% RSLogix 500 project Temperature Control and Alarm System.RSS, saved by version 8.30.00.16 %
PROJECT "UNTITLED"    % processor: Bul.1763 MicroLogix 1100 Series B %

PROGRAM FILES
  LAD 2 "MAIN"  9 rungs
  LAD 3 "DIGITAL IO"  10 rungs
  LAD 4 "ANALOG IO"  4 rungs
  LAD 5 "MANUAL"  10 rungs
  LAD 6 "AUTOMATIC"  3 rungs
  LAD 7 "ALARMS"  13 rungs
  LAD 8 "TEMP PID"  10 rungs
  LAD 9 "PROCESS"  9 rungs
  LAD 10 "TIMERS"  7 rungs

DATA FILES
  O0 OUTPUT  4 elements
  I1 INPUT  6 elements
  S2 STATUS  66 elements
  B3 BINARY  3 elements
  T4 TIMER  6 elements
  C5 COUNTER  1 elements
  R6 CONTROL  1 elements
  N7 INTEGER  5 elements
  F8 FLOAT  6 elements

LADDER 2 "MAIN"
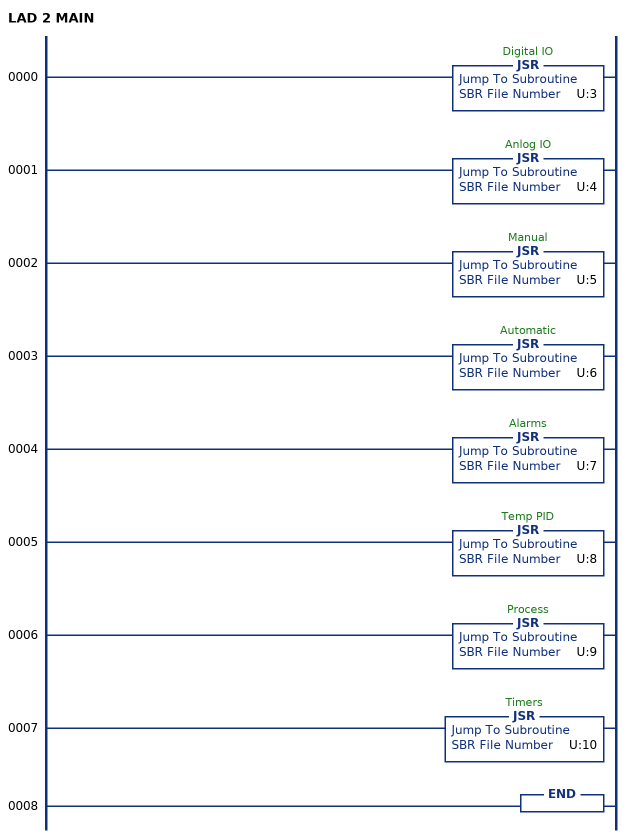
% Rung: 0 %
SOR JSR U:3 EOR
%   U:3  "Digital IO" %
% Rung: 1 %
SOR JSR U:4 EOR
%   U:4  "Anlog IO" %
% Rung: 2 %
SOR JSR U:5 EOR
%   U:5  "Manual" %
% Rung: 3 %
SOR JSR U:6 EOR
%   U:6  "Automatic" %
% Rung: 4 %
SOR JSR U:7 EOR
%   U:7  "Alarms" %
% Rung: 5 %
SOR JSR U:8 EOR
%   U:8  "Temp PID" %
% Rung: 6 %
SOR JSR U:9 EOR
%   U:9  "Process" %
% Rung: 7 %
SOR JSR U:10 EOR
%   U:10  "Timers" %
% Rung: 8 %
SOR END EOR

LADDER 3 "DIGITAL IO"
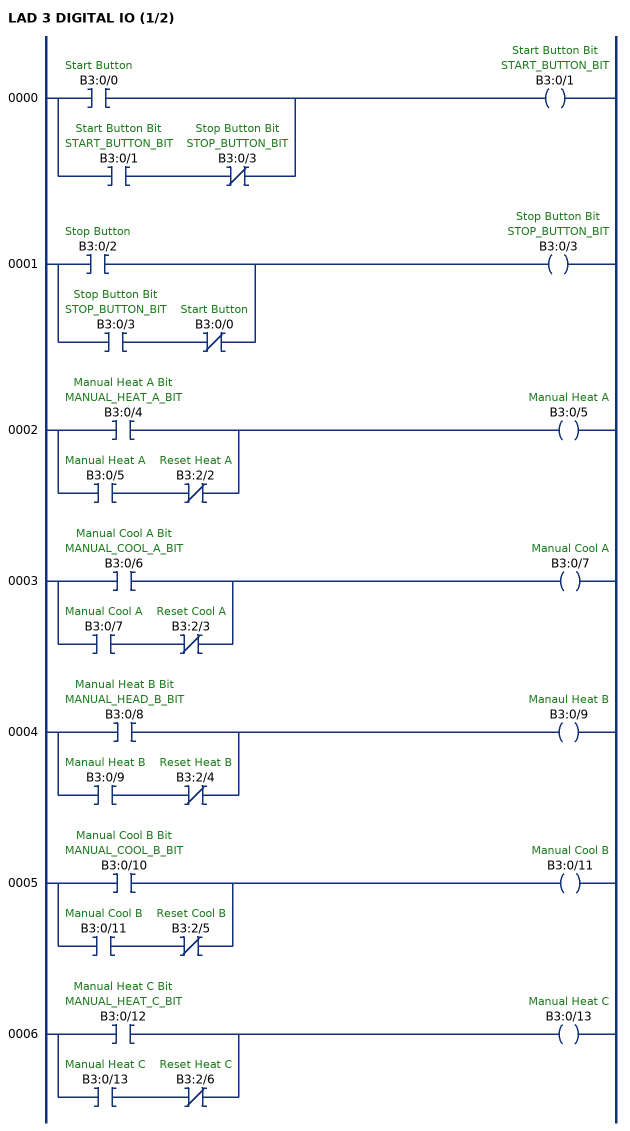
% Rung: 0 %
SOR BST XIC B3:0/0 NXB XIC B3:0/1 XIO B3:0/3 BND OTE B3:0/1 EOR
%   B3:0/0  "Start Button" %
%   B3:0/1  START_BUTTON_BIT  "Start Button Bit" %
%   B3:0/3  STOP_BUTTON_BIT  "Stop Button Bit" %
% Rung: 1 %
SOR BST XIC B3:0/2 NXB XIC B3:0/3 XIO B3:0/0 BND OTE B3:0/3 EOR
%   B3:0/2  "Stop Button" %
%   B3:0/3  STOP_BUTTON_BIT  "Stop Button Bit" %
%   B3:0/0  "Start Button" %
% Rung: 2 %
SOR BST XIC B3:0/4 NXB XIC B3:0/5 XIO B3:2/2 BND OTE B3:0/5 EOR
%   B3:0/4  MANUAL_HEAT_A_BIT  "Manual Heat A Bit" %
%   B3:0/5  "Manual Heat A" %
%   B3:2/2  "Reset Heat A" %
% Rung: 3 %
SOR BST XIC B3:0/6 NXB XIC B3:0/7 XIO B3:2/3 BND OTE B3:0/7 EOR
%   B3:0/6  MANUAL_COOL_A_BIT  "Manual Cool A Bit" %
%   B3:0/7  "Manual Cool A" %
%   B3:2/3  "Reset Cool A" %
% Rung: 4 %
SOR BST XIC B3:0/8 NXB XIC B3:0/9 XIO B3:2/4 BND OTE B3:0/9 EOR
%   B3:0/8  MANUAL_HEAD_B_BIT  "Manual Heat B Bit" %
%   B3:0/9  "Manaul Heat B" %
%   B3:2/4  "Reset Heat B" %
% Rung: 5 %
SOR BST XIC B3:0/10 NXB XIC B3:0/11 XIO B3:2/5 BND OTE B3:0/11 EOR
%   B3:0/10  MANUAL_COOL_B_BIT  "Manual Cool B Bit" %
%   B3:0/11  "Manual Cool B" %
%   B3:2/5  "Reset Cool B" %
% Rung: 6 %
SOR BST XIC B3:0/12 NXB XIC B3:0/13 XIO B3:2/6 BND OTE B3:0/13 EOR
%   B3:0/12  MANUAL_HEAT_C_BIT  "Manual Heat C Bit" %
%   B3:0/13  "Manual Heat C" %
%   B3:2/6  "Reset Heat C" %

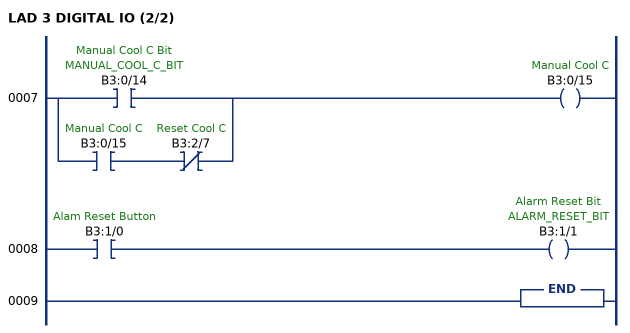
% Rung: 7 %
SOR BST XIC B3:0/14 NXB XIC B3:0/15 XIO B3:2/7 BND OTE B3:0/15 EOR
%   B3:0/14  MANUAL_COOL_C_BIT  "Manual Cool C Bit" %
%   B3:0/15  "Manual Cool C" %
%   B3:2/7  "Reset Cool C" %
% Rung: 8 %
SOR XIC B3:1/0 OTE B3:1/1 EOR
%   B3:1/0  "Alam Reset Button" %
%   B3:1/1  ALARM_RESET_BIT  "Alarm Reset Bit" %
% Rung: 9 %
SOR END EOR

LADDER 4 "ANALOG IO"
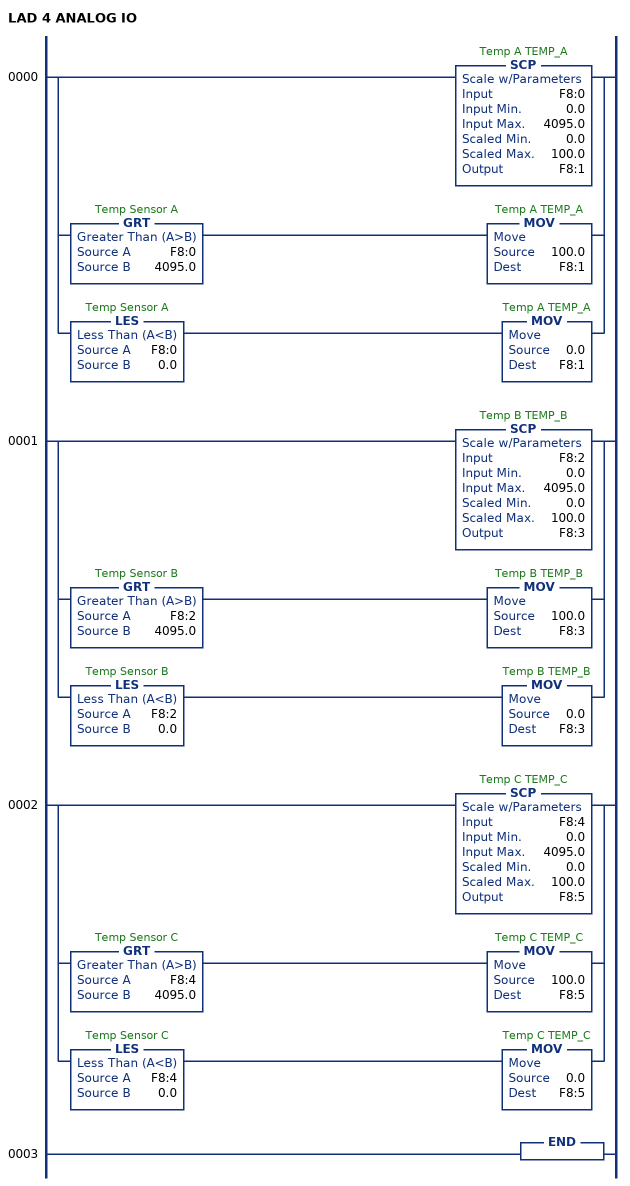
% Rung: 0 %
SOR BST BST SCP F8:0 0.0 4095.0 0.0 100.0 F8:1 NXB GRT F8:0 4095.0 MOV 100.0 F8:1 BND NXB LES F8:0 0.0 MOV 0.0 F8:1 BND EOR
%   F8:0  "Temp Sensor A" %
%   F8:1  TEMP_A  "Temp A" %
% Rung: 1 %
SOR BST BST SCP F8:2 0.0 4095.0 0.0 100.0 F8:3 NXB GRT F8:2 4095.0 MOV 100.0 F8:3 BND NXB LES F8:2 0.0 MOV 0.0 F8:3 BND EOR
%   F8:2  "Temp Sensor B" %
%   F8:3  TEMP_B  "Temp B" %
% Rung: 2 %
SOR BST BST SCP F8:4 0.0 4095.0 0.0 100.0 F8:5 NXB GRT F8:4 4095.0 MOV 100.0 F8:5 BND NXB LES F8:4 0.0 MOV 0.0 F8:5 BND EOR
%   F8:4  "Temp Sensor C" %
%   F8:5  TEMP_C  "Temp C" %
% Rung: 3 %
SOR END EOR

LADDER 5 "MANUAL"
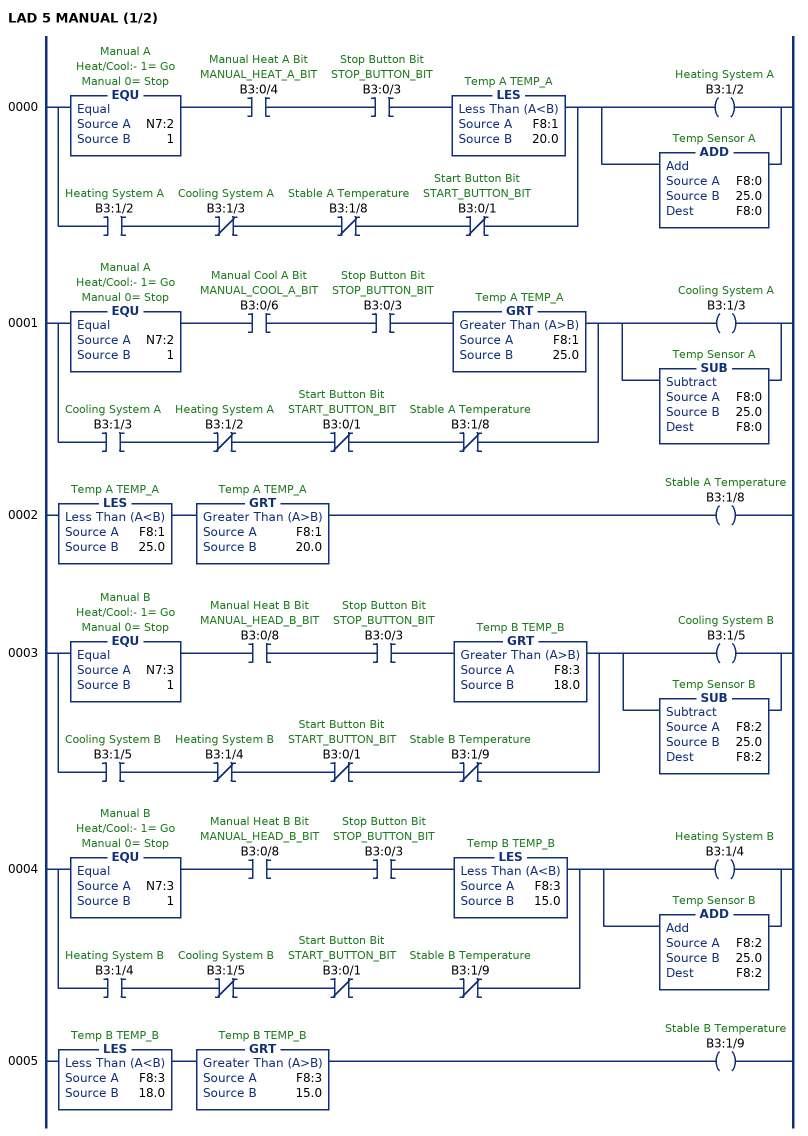
% Rung: 0 %
SOR BST EQU N7:2 1 XIC B3:0/4 XIC B3:0/3 LES F8:1 20.0 NXB XIC B3:1/2 XIO B3:1/3 XIO B3:1/8 XIO B3:0/1 BND BST OTE B3:1/2 NXB ADD F8:0 25.0 F8:0 BND EOR
%   N7:2  "Manual A Heat/Cool:- 1= Go Manual 0= Stop" %
%   B3:0/4  MANUAL_HEAT_A_BIT  "Manual Heat A Bit" %
%   B3:0/3  STOP_BUTTON_BIT  "Stop Button Bit" %
%   F8:1  TEMP_A  "Temp A" %
%   B3:1/2  "Heating System A" %
%   B3:1/3  "Cooling System A" %
%   B3:1/8  "Stable A Temperature" %
%   B3:0/1  START_BUTTON_BIT  "Start Button Bit" %
%   F8:0  "Temp Sensor A" %
% Rung: 1 %
SOR BST EQU N7:2 1 XIC B3:0/6 XIC B3:0/3 GRT F8:1 25.0 NXB XIC B3:1/3 XIO B3:1/2 XIO B3:0/1 XIO B3:1/8 BND BST OTE B3:1/3 NXB SUB F8:0 25.0 F8:0 BND EOR
%   N7:2  "Manual A Heat/Cool:- 1= Go Manual 0= Stop" %
%   B3:0/6  MANUAL_COOL_A_BIT  "Manual Cool A Bit" %
%   B3:0/3  STOP_BUTTON_BIT  "Stop Button Bit" %
%   F8:1  TEMP_A  "Temp A" %
%   B3:1/3  "Cooling System A" %
%   B3:1/2  "Heating System A" %
%   B3:0/1  START_BUTTON_BIT  "Start Button Bit" %
%   B3:1/8  "Stable A Temperature" %
%   F8:0  "Temp Sensor A" %
% Rung: 2 %
SOR LES F8:1 25.0 GRT F8:1 20.0 OTE B3:1/8 EOR
%   F8:1  TEMP_A  "Temp A" %
%   B3:1/8  "Stable A Temperature" %
% Rung: 3 %
SOR BST EQU N7:3 1 XIC B3:0/8 XIC B3:0/3 GRT F8:3 18.0 NXB XIC B3:1/5 XIO B3:1/4 XIO B3:0/1 XIO B3:1/9 BND BST OTE B3:1/5 NXB SUB F8:2 25.0 F8:2 BND EOR
%   N7:3  "Manual B Heat/Cool:- 1= Go Manual 0= Stop" %
%   B3:0/8  MANUAL_HEAD_B_BIT  "Manual Heat B Bit" %
%   B3:0/3  STOP_BUTTON_BIT  "Stop Button Bit" %
%   F8:3  TEMP_B  "Temp B" %
%   B3:1/5  "Cooling System B" %
%   B3:1/4  "Heating System B" %
%   B3:0/1  START_BUTTON_BIT  "Start Button Bit" %
%   B3:1/9  "Stable B Temperature" %
%   F8:2  "Temp Sensor B" %
% Rung: 4 %
SOR BST EQU N7:3 1 XIC B3:0/8 XIC B3:0/3 LES F8:3 15.0 NXB XIC B3:1/4 XIO B3:1/5 XIO B3:0/1 XIO B3:1/9 BND BST OTE B3:1/4 NXB ADD F8:2 25.0 F8:2 BND EOR
%   N7:3  "Manual B Heat/Cool:- 1= Go Manual 0= Stop" %
%   B3:0/8  MANUAL_HEAD_B_BIT  "Manual Heat B Bit" %
%   B3:0/3  STOP_BUTTON_BIT  "Stop Button Bit" %
%   F8:3  TEMP_B  "Temp B" %
%   B3:1/4  "Heating System B" %
%   B3:1/5  "Cooling System B" %
%   B3:0/1  START_BUTTON_BIT  "Start Button Bit" %
%   B3:1/9  "Stable B Temperature" %
%   F8:2  "Temp Sensor B" %
% Rung: 5 %
SOR LES F8:3 18.0 GRT F8:3 15.0 OTE B3:1/9 EOR
%   F8:3  TEMP_B  "Temp B" %
%   B3:1/9  "Stable B Temperature" %

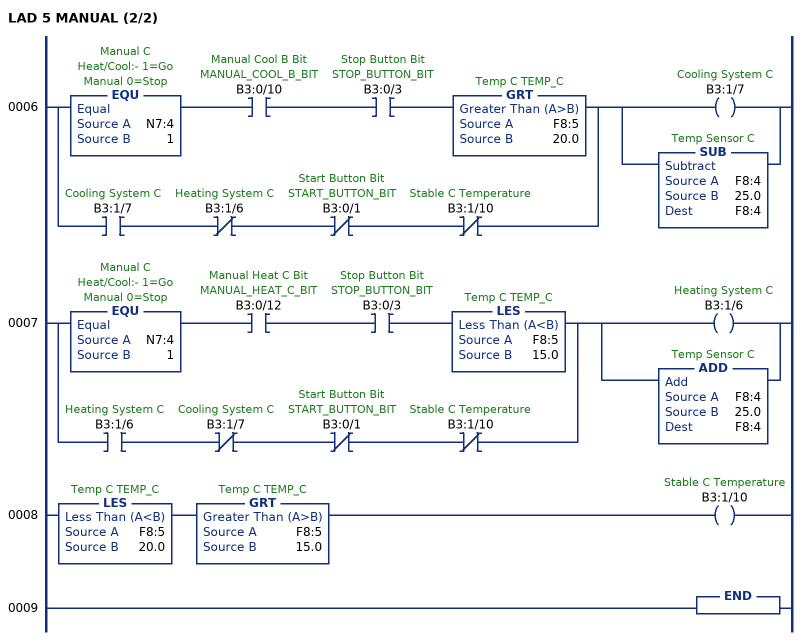
% Rung: 6 %
SOR BST EQU N7:4 1 XIC B3:0/10 XIC B3:0/3 GRT F8:5 20.0 NXB XIC B3:1/7 XIO B3:1/6 XIO B3:0/1 XIO B3:1/10 BND BST OTE B3:1/7 NXB SUB F8:4 25.0 F8:4 BND EOR
%   N7:4  "Manual C Heat/Cool:- 1=Go Manual 0=Stop" %
%   B3:0/10  MANUAL_COOL_B_BIT  "Manual Cool B Bit" %
%   B3:0/3  STOP_BUTTON_BIT  "Stop Button Bit" %
%   F8:5  TEMP_C  "Temp C" %
%   B3:1/7  "Cooling System C" %
%   B3:1/6  "Heating System C" %
%   B3:0/1  START_BUTTON_BIT  "Start Button Bit" %
%   B3:1/10  "Stable C Temperature" %
%   F8:4  "Temp Sensor C" %
% Rung: 7 %
SOR BST EQU N7:4 1 XIC B3:0/12 XIC B3:0/3 LES F8:5 15.0 NXB XIC B3:1/6 XIO B3:1/7 XIO B3:0/1 XIO B3:1/10 BND BST OTE B3:1/6 NXB ADD F8:4 25.0 F8:4 BND EOR
%   N7:4  "Manual C Heat/Cool:- 1=Go Manual 0=Stop" %
%   B3:0/12  MANUAL_HEAT_C_BIT  "Manual Heat C Bit" %
%   B3:0/3  STOP_BUTTON_BIT  "Stop Button Bit" %
%   F8:5  TEMP_C  "Temp C" %
%   B3:1/6  "Heating System C" %
%   B3:1/7  "Cooling System C" %
%   B3:0/1  START_BUTTON_BIT  "Start Button Bit" %
%   B3:1/10  "Stable C Temperature" %
%   F8:4  "Temp Sensor C" %
% Rung: 8 %
SOR LES F8:5 20.0 GRT F8:5 15.0 OTE B3:1/10 EOR
%   F8:5  TEMP_C  "Temp C" %
%   B3:1/10  "Stable C Temperature" %
% Rung: 9 %
SOR END EOR

LADDER 6 "AUTOMATIC"
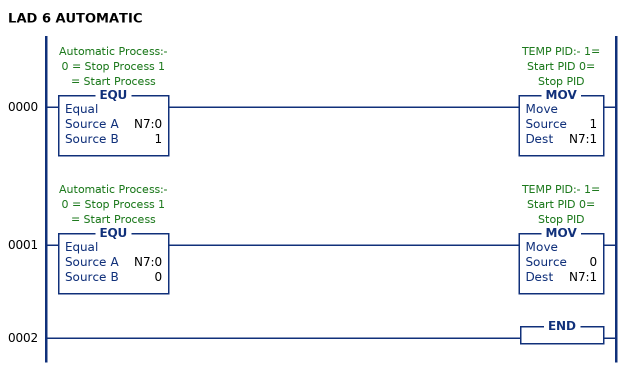
% Rung: 0 %
SOR EQU N7:0 1 MOV 1 N7:1 EOR
%   N7:0  "Automatic Process:- 0 = Stop Process 1 = Start Process" %
%   N7:1  "TEMP PID:- 1= Start PID 0= Stop PID" %
% Rung: 1 %
SOR EQU N7:0 0 MOV 0 N7:1 EOR
%   N7:0  "Automatic Process:- 0 = Stop Process 1 = Start Process" %
%   N7:1  "TEMP PID:- 1= Start PID 0= Stop PID" %
% Rung: 2 %
SOR END EOR

LADDER 7 "ALARMS"
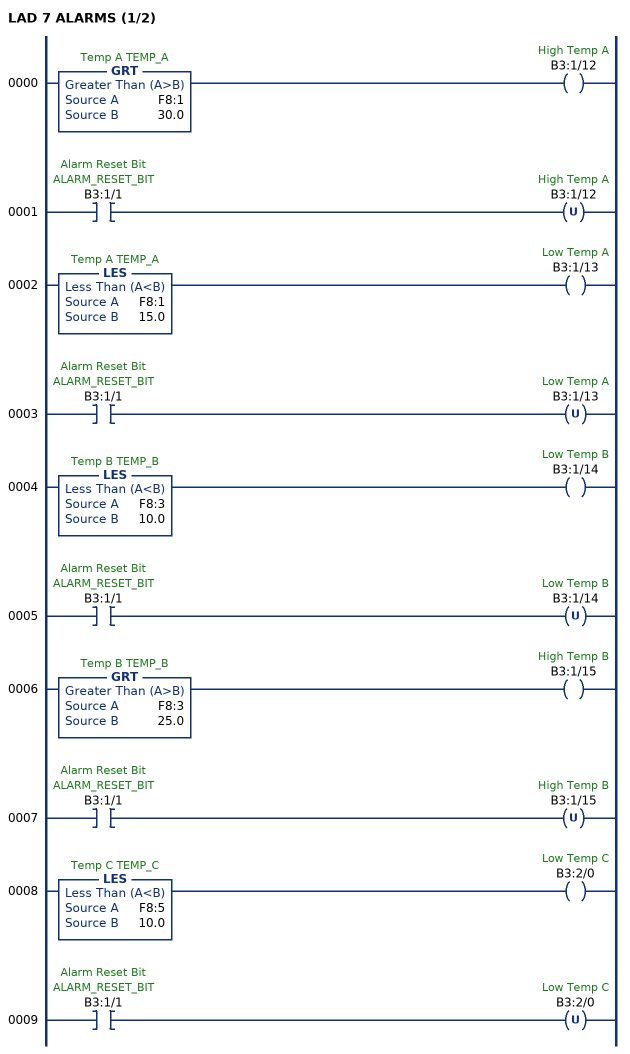
% Rung: 0 %
SOR GRT F8:1 30.0 OTE B3:1/12 EOR
%   F8:1  TEMP_A  "Temp A" %
%   B3:1/12  "High Temp A" %
% Rung: 1 %
SOR XIC B3:1/1 OTU B3:1/12 EOR
%   B3:1/1  ALARM_RESET_BIT  "Alarm Reset Bit" %
%   B3:1/12  "High Temp A" %
% Rung: 2 %
SOR LES F8:1 15.0 OTE B3:1/13 EOR
%   F8:1  TEMP_A  "Temp A" %
%   B3:1/13  "Low Temp A" %
% Rung: 3 %
SOR XIC B3:1/1 OTU B3:1/13 EOR
%   B3:1/1  ALARM_RESET_BIT  "Alarm Reset Bit" %
%   B3:1/13  "Low Temp A" %
% Rung: 4 %
SOR LES F8:3 10.0 OTE B3:1/14 EOR
%   F8:3  TEMP_B  "Temp B" %
%   B3:1/14  "Low Temp B" %
% Rung: 5 %
SOR XIC B3:1/1 OTU B3:1/14 EOR
%   B3:1/1  ALARM_RESET_BIT  "Alarm Reset Bit" %
%   B3:1/14  "Low Temp B" %
% Rung: 6 %
SOR GRT F8:3 25.0 OTE B3:1/15 EOR
%   F8:3  TEMP_B  "Temp B" %
%   B3:1/15  "High Temp B" %
% Rung: 7 %
SOR XIC B3:1/1 OTU B3:1/15 EOR
%   B3:1/1  ALARM_RESET_BIT  "Alarm Reset Bit" %
%   B3:1/15  "High Temp B" %
% Rung: 8 %
SOR LES F8:5 10.0 OTE B3:2/0 EOR
%   F8:5  TEMP_C  "Temp C" %
%   B3:2/0  "Low Temp C" %
% Rung: 9 %
SOR XIC B3:1/1 OTU B3:2/0 EOR
%   B3:1/1  ALARM_RESET_BIT  "Alarm Reset Bit" %
%   B3:2/0  "Low Temp C" %

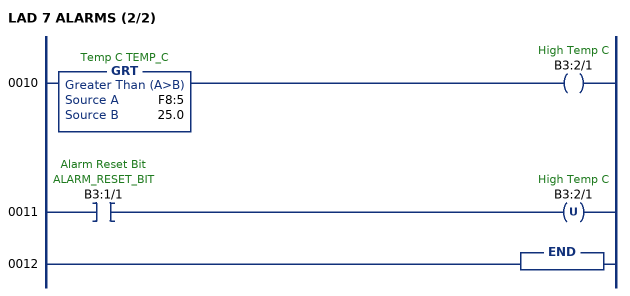
% Rung: 10 %
SOR GRT F8:5 25.0 OTE B3:2/1 EOR
%   F8:5  TEMP_C  "Temp C" %
%   B3:2/1  "High Temp C" %
% Rung: 11 %
SOR XIC B3:1/1 OTU B3:2/1 EOR
%   B3:1/1  ALARM_RESET_BIT  "Alarm Reset Bit" %
%   B3:2/1  "High Temp C" %
% Rung: 12 %
SOR END EOR

LADDER 8 "TEMP PID"
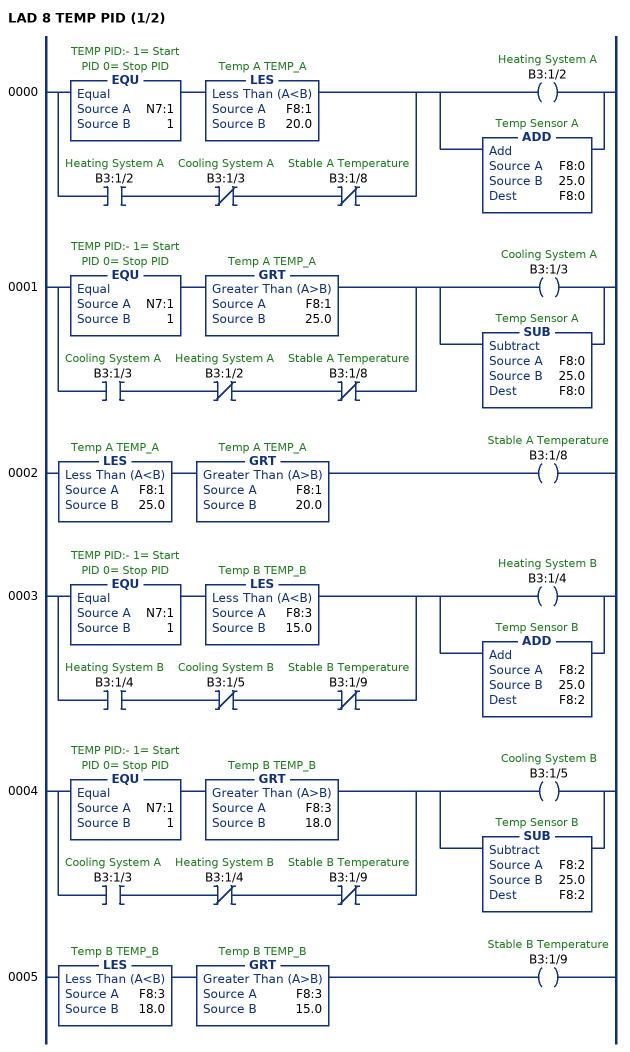
% Rung: 0 %
SOR BST EQU N7:1 1 LES F8:1 20.0 NXB XIC B3:1/2 XIO B3:1/3 XIO B3:1/8 BND BST OTE B3:1/2 NXB ADD F8:0 25.0 F8:0 BND EOR
%   N7:1  "TEMP PID:- 1= Start PID 0= Stop PID" %
%   F8:1  TEMP_A  "Temp A" %
%   B3:1/2  "Heating System A" %
%   B3:1/3  "Cooling System A" %
%   B3:1/8  "Stable A Temperature" %
%   F8:0  "Temp Sensor A" %
% Rung: 1 %
SOR BST EQU N7:1 1 GRT F8:1 25.0 NXB XIC B3:1/3 XIO B3:1/2 XIO B3:1/8 BND BST OTE B3:1/3 NXB SUB F8:0 25.0 F8:0 BND EOR
%   N7:1  "TEMP PID:- 1= Start PID 0= Stop PID" %
%   F8:1  TEMP_A  "Temp A" %
%   B3:1/3  "Cooling System A" %
%   B3:1/2  "Heating System A" %
%   B3:1/8  "Stable A Temperature" %
%   F8:0  "Temp Sensor A" %
% Rung: 2 %
SOR LES F8:1 25.0 GRT F8:1 20.0 OTE B3:1/8 EOR
%   F8:1  TEMP_A  "Temp A" %
%   B3:1/8  "Stable A Temperature" %
% Rung: 3 %
SOR BST EQU N7:1 1 LES F8:3 15.0 NXB XIC B3:1/4 XIO B3:1/5 XIO B3:1/9 BND BST OTE B3:1/4 NXB ADD F8:2 25.0 F8:2 BND EOR
%   N7:1  "TEMP PID:- 1= Start PID 0= Stop PID" %
%   F8:3  TEMP_B  "Temp B" %
%   B3:1/4  "Heating System B" %
%   B3:1/5  "Cooling System B" %
%   B3:1/9  "Stable B Temperature" %
%   F8:2  "Temp Sensor B" %
% Rung: 4 %
SOR BST EQU N7:1 1 GRT F8:3 18.0 NXB XIC B3:1/3 XIO B3:1/4 XIO B3:1/9 BND BST OTE B3:1/5 NXB SUB F8:2 25.0 F8:2 BND EOR
%   N7:1  "TEMP PID:- 1= Start PID 0= Stop PID" %
%   F8:3  TEMP_B  "Temp B" %
%   B3:1/3  "Cooling System A" %
%   B3:1/4  "Heating System B" %
%   B3:1/9  "Stable B Temperature" %
%   B3:1/5  "Cooling System B" %
%   F8:2  "Temp Sensor B" %
% Rung: 5 %
SOR LES F8:3 18.0 GRT F8:3 15.0 OTE B3:1/9 EOR
%   F8:3  TEMP_B  "Temp B" %
%   B3:1/9  "Stable B Temperature" %

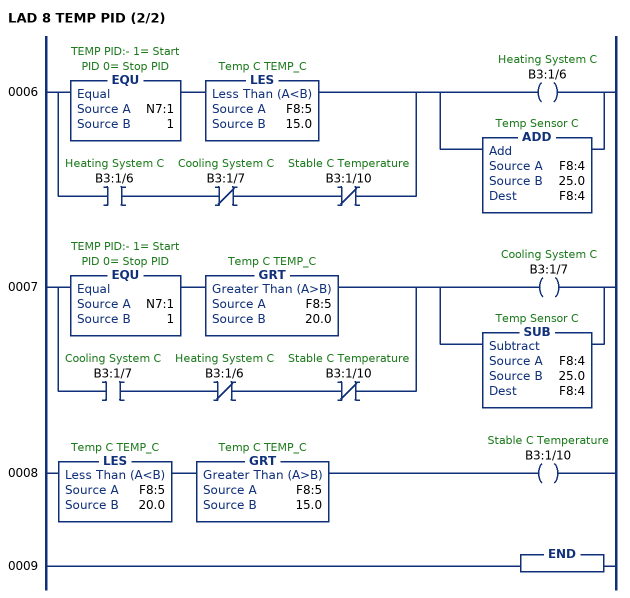
% Rung: 6 %
SOR BST EQU N7:1 1 LES F8:5 15.0 NXB XIC B3:1/6 XIO B3:1/7 XIO B3:1/10 BND BST OTE B3:1/6 NXB ADD F8:4 25.0 F8:4 BND EOR
%   N7:1  "TEMP PID:- 1= Start PID 0= Stop PID" %
%   F8:5  TEMP_C  "Temp C" %
%   B3:1/6  "Heating System C" %
%   B3:1/7  "Cooling System C" %
%   B3:1/10  "Stable C Temperature" %
%   F8:4  "Temp Sensor C" %
% Rung: 7 %
SOR BST EQU N7:1 1 GRT F8:5 20.0 NXB XIC B3:1/7 XIO B3:1/6 XIO B3:1/10 BND BST OTE B3:1/7 NXB SUB F8:4 25.0 F8:4 BND EOR
%   N7:1  "TEMP PID:- 1= Start PID 0= Stop PID" %
%   F8:5  TEMP_C  "Temp C" %
%   B3:1/7  "Cooling System C" %
%   B3:1/6  "Heating System C" %
%   B3:1/10  "Stable C Temperature" %
%   F8:4  "Temp Sensor C" %
% Rung: 8 %
SOR LES F8:5 20.0 GRT F8:5 15.0 OTE B3:1/10 EOR
%   F8:5  TEMP_C  "Temp C" %
%   B3:1/10  "Stable C Temperature" %
% Rung: 9 %
SOR END EOR

LADDER 9 "PROCESS"
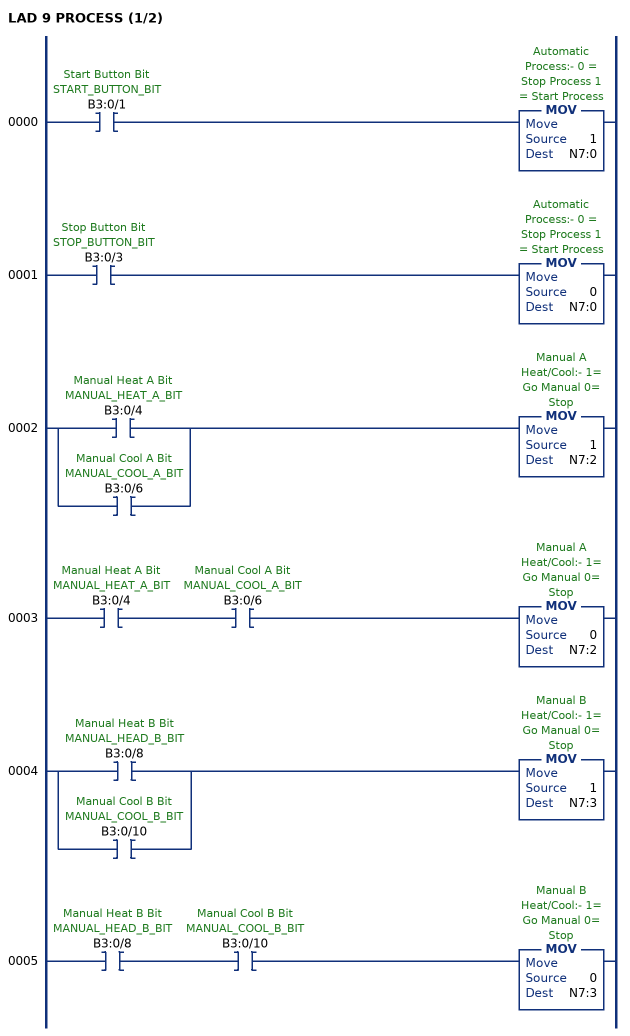
% Rung: 0 %
SOR XIC B3:0/1 MOV 1 N7:0 EOR
%   B3:0/1  START_BUTTON_BIT  "Start Button Bit" %
%   N7:0  "Automatic Process:- 0 = Stop Process 1 = Start Process" %
% Rung: 1 %
SOR XIC B3:0/3 MOV 0 N7:0 EOR
%   B3:0/3  STOP_BUTTON_BIT  "Stop Button Bit" %
%   N7:0  "Automatic Process:- 0 = Stop Process 1 = Start Process" %
% Rung: 2 %
SOR BST XIC B3:0/4 NXB XIC B3:0/6 BND MOV 1 N7:2 EOR
%   B3:0/4  MANUAL_HEAT_A_BIT  "Manual Heat A Bit" %
%   B3:0/6  MANUAL_COOL_A_BIT  "Manual Cool A Bit" %
%   N7:2  "Manual A Heat/Cool:- 1= Go Manual 0= Stop" %
% Rung: 3 %
SOR XIC B3:0/4 XIC B3:0/6 MOV 0 N7:2 EOR
%   B3:0/4  MANUAL_HEAT_A_BIT  "Manual Heat A Bit" %
%   B3:0/6  MANUAL_COOL_A_BIT  "Manual Cool A Bit" %
%   N7:2  "Manual A Heat/Cool:- 1= Go Manual 0= Stop" %
% Rung: 4 %
SOR BST XIC B3:0/8 NXB XIC B3:0/10 BND MOV 1 N7:3 EOR
%   B3:0/8  MANUAL_HEAD_B_BIT  "Manual Heat B Bit" %
%   B3:0/10  MANUAL_COOL_B_BIT  "Manual Cool B Bit" %
%   N7:3  "Manual B Heat/Cool:- 1= Go Manual 0= Stop" %
% Rung: 5 %
SOR XIC B3:0/8 XIC B3:0/10 MOV 0 N7:3 EOR
%   B3:0/8  MANUAL_HEAD_B_BIT  "Manual Heat B Bit" %
%   B3:0/10  MANUAL_COOL_B_BIT  "Manual Cool B Bit" %
%   N7:3  "Manual B Heat/Cool:- 1= Go Manual 0= Stop" %

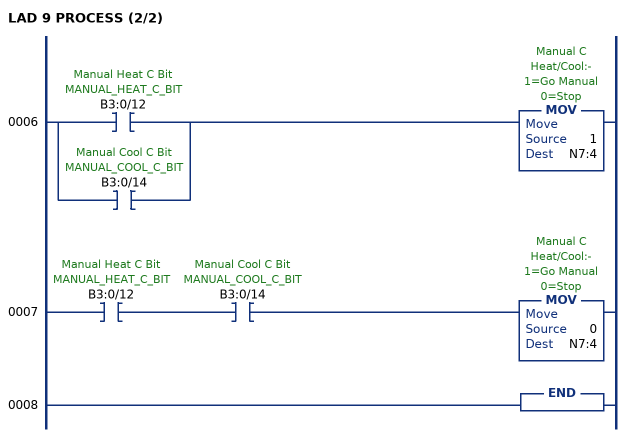
% Rung: 6 %
SOR BST XIC B3:0/12 NXB XIC B3:0/14 BND MOV 1 N7:4 EOR
%   B3:0/12  MANUAL_HEAT_C_BIT  "Manual Heat C Bit" %
%   B3:0/14  MANUAL_COOL_C_BIT  "Manual Cool C Bit" %
%   N7:4  "Manual C Heat/Cool:- 1=Go Manual 0=Stop" %
% Rung: 7 %
SOR XIC B3:0/12 XIC B3:0/14 MOV 0 N7:4 EOR
%   B3:0/12  MANUAL_HEAT_C_BIT  "Manual Heat C Bit" %
%   B3:0/14  MANUAL_COOL_C_BIT  "Manual Cool C Bit" %
%   N7:4  "Manual C Heat/Cool:- 1=Go Manual 0=Stop" %
% Rung: 8 %
SOR END EOR

LADDER 10 "TIMERS"
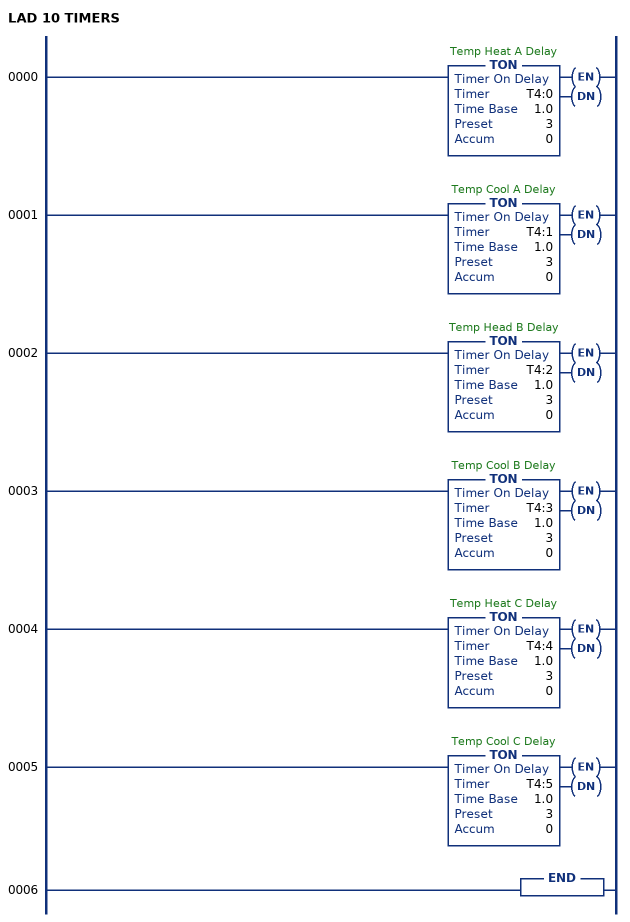
% Rung: 0 %
SOR TON T4:0 1.0 3 0 EOR
%   T4:0  "Temp Heat A Delay" %
% Rung: 1 %
SOR TON T4:1 1.0 3 0 EOR
%   T4:1  "Temp Cool A Delay" %
% Rung: 2 %
SOR TON T4:2 1.0 3 0 EOR
%   T4:2  "Temp Head B Delay" %
% Rung: 3 %
SOR TON T4:3 1.0 3 0 EOR
%   T4:3  "Temp Cool B Delay" %
% Rung: 4 %
SOR TON T4:4 1.0 3 0 EOR
%   T4:4  "Temp Heat C Delay" %
% Rung: 5 %
SOR TON T4:5 1.0 3 0 EOR
%   T4:5  "Temp Cool C Delay" %
% Rung: 6 %
SOR END EOR

OTHER DOCUMENTED ADDRESSES
  B3:1/11  "One Shot"
  T4:0/DN  "Heat A DN"
  T4:0/EN  "Heat A EN"

DATA TABLE (non-zero values as saved)
DATA T4
% .PRE .ACC %
% T4:0 % 3 0
% T4:1 % 3 0
% T4:2 % 3 0
% T4:3 % 3 0
% T4:4 % 3 0
% T4:5 % 3 0
